(* IEC 61131-3 sources: AXOpen/src/timers/ctrl/test, 4 files *)

(* ---- Abstractions.st ---- *)
USING AxUnit;
USING AXOpen.Timers;
USING AXOpen.Rtc;
USING AXOpen.Logging;
USING AXOpen.Core;
USING AXOpen.Rtc;
USING AXOpen.Rtm;

NAMESPACE AXOpen.Timers_tests

    {S7.extern=ReadWrite}
    CLASS INTERNAL _NULL_LOGGER IMPLEMENTS IAxoLogger
        METHOD PUBLIC Log
            VAR_INPUT
                _message : STRING[80];
                _level : eLogLevel;
                _sender : IAxoObject;
            END_VAR
            ;
        END_METHOD

        METHOD PUBLIC Log
            VAR_INPUT
                _message : STRING[80];
                _level : eLogLevel;
            END_VAR
            ;
        END_METHOD

        METHOD PUBLIC SetMinimumLevel : IAxoLoggerConfig
            VAR_INPUT
                _level : eLogLevel;
            END_VAR
            ;
        END_METHOD
    END_CLASS

    {S7.extern=ReadWrite}
    CLASS INTERNAL AxoRtmMock IMPLEMENTS IAxoRtm
        VAR PRIVATE
            _elapsed : LTIME;
        END_VAR

        METHOD INTERNAL SetElapsed : LDATE_AND_TIME
            VAR_INPUT
                Set :  LTIME;
            END_VAR;
            _elapsed := Set;
        END_METHOD

        METHOD PUBLIC Elapsed : LTIME
            Elapsed := _elapsed;
        END_METHOD
    END_CLASS

    {S7.extern=ReadWrite}
    CLASS INTERNAL TestContext IMPLEMENTS IAxoContext
        VAR PROTECTED
            _openCounter : ULINT;
            _closeCounter : ULINT;
            _identityCounter : ULINT;
            _rtc :  IAxoRtc;
            _rtm :  IAxoRtm;
         END_VAR
        METHOD PUBLIC Open : ULINT
            _openCounter := _openCounter + ULINT#1;
        END_METHOD

        METHOD PUBLIC Close : ULINT
            _closeCounter := _closeCounter + ULINT#1;
        END_METHOD

        METHOD PUBLIC OpenCycleCount : ULINT
            OpenCycleCount := _openCounter;
        END_METHOD

        METHOD PUBLIC ClosedCycleCount : ULINT
            ClosedCycleCount := _closeCounter;
        END_METHOD

        METHOD PUBLIC CreateIdentity : ULINT
            _identityCounter := _identityCounter + ULINT#1;
            CreateIdentity := _identityCounter;
        END_METHOD

        METHOD PUBLIC GetRtc : IAxoRtc ;
            GetRtc := _rtc;
        END_METHOD

        METHOD PUBLIC InjectRtc
             VAR_INPUT Rtc : IAxoRtc;
            END_VAR ;

            _rtc := Rtc;
        END_METHOD

        VAR PRIVATE
            NULL_LOGGER : _NULL_LOGGER;
        END_VAR
        METHOD PUBLIC GetLogger : AXOpen.Logging.IAxoLogger GetLogger := NULL_LOGGER; END_METHOD
        METHOD PUBLIC InjectLogger VAR_INPUT _logger : AXOpen.Logging.IAxoLogger; END_VAR ; END_METHOD

        METHOD PUBLIC GetRtm : IAxoRtm GetRtm := _rtm; END_METHOD
        METHOD PUBLIC InjectRtm VAR_INPUT inRtm : IAxoRtm; END_VAR _rtm := inRtm; END_METHOD
    END_CLASS
END_NAMESPACE

(* ---- OffDelayTests.st ---- *)
USING AxUnit;
USING AXOpen.Timers;
USING AXOpen.Rtc;
USING AXOpen.Logging;
USING AXOpen.Core;
USING AXOpen.Rtc;

NAMESPACE AXOpen.Timers_tests

    {TestFixture}
    {S7.extern=ReadWrite}
    CLASS AxoOffDelayTimersTests
        VAR PROTECTED
            _context : TestContext;
            _inspectedBool : BOOL;
            _rtcMock :  AxoRtmMock;
            _signal : BOOL;
            _testTimerOnDelay: AXOpen.Timers.OnDelayTimer;
            _testTimerOffDelay: AXOpen.Timers.OffDelayTimer;
            _testTimeDelay: LTIME := LTIME#5s;
        END_VAR

        METHOD PRIVATE Initialize
            _context.InjectRtm(_rtcMock);
        END_METHOD

        VAR
            _contextBlank : TestContext;
            _testTimerOnDelayBlank: AXOpen.Timers.OnDelayTimer;
            _testTimerOffDelayBlank: AXOpen.Timers.OffDelayTimer;
        END_VAR

        {TestSetup}
        METHOD PUBLIC TestSetup
        // Will be called before MyTest_A AND before Test_B are executed
            _context := _contextBlank;
            _testTimerOnDelay := _testTimerOnDelayBlank;
            _testTimerOffDelay := _testTimerOffDelayBlank;
        END_METHOD

        {TestTearDown}
        METHOD PUBLIC TestTearDown
        // Will be called after MyTest_A AND before Test_B where executed
            ;
        END_METHOD

        {FixtureSetup}
        METHOD PUBLIC FixtureSetup
        // Will be called once before the Tests are executed
            ;
        END_METHOD

        {FixtureTearDown}
        METHOD PUBLIC FixtureTearDown
        // Will be called after the Tests where executed
            ;
        END_METHOD

        {Test}
        METHOD PUBLIC Timer_offDelay_class_output_test
            THIS.Initialize();

            _context.Open();

            //_rtcMock.SetElapsed(LT#1980-01-23-13:14:33.123456);
            _rtcMock.SetElapsed(LT#0S);
            _signal := TRUE;
            _testTimerOffDelay.OffDelay(_context, _signal, _testTimeDelay);
            Assert.Equal(TRUE, _testTimerOffDelay.output);

            //move 6 seconds in future, timer stil don't count, true is output
            //_rtcMock.SetNowUTC(LDT#1980-01-23-13:14:39.123456);
            _rtcMock.SetElapsed(LT#6S);
            _testTimerOffDelay.OffDelay(_context, _signal, _testTimeDelay);
            Assert.Equal(TRUE, _testTimerOffDelay.output);

            //here, timer starts count
            //_rtcMock.SetNowUTC(LDT#1980-01-23-13:14:41.123456);
            _rtcMock.SetElapsed(LT#9S);
            _signal := FALSE;
            _testTimerOffDelay.OffDelay(_context, _signal, _testTimeDelay);
            Assert.Equal(TRUE, _testTimerOffDelay.output);

            //here, timer should hit delay and turn off signal
            //_rtcMock.SetNowUTC(LDT#1980-01-23-13:14:46.123456);
            _rtcMock.SetElapsed(LT#14S);
            _testTimerOffDelay.OffDelay(_context, _signal, _testTimeDelay);
            Assert.Equal(FALSE, _testTimerOffDelay.output);

            _context.Close();
        END_METHOD

        {Test}
        METHOD PUBLIC Timer_offDelay_overall_test
            THIS.Initialize();

            _context.Open();

            //all turn off, previous signal was false, input is false, output should be false
            //_rtcMock.SetNowUTC(LDT#1980-01-23-13:14:30.0);
            _rtcMock.SetElapsed(LT#10S);
            _signal := FALSE;
            _testTimerOffDelay.OffDelay(_context, _signal, _testTimeDelay);
            Assert.Equal(FALSE, _testTimerOffDelay.output);

            //after 1 second, turn on signal, output should be on
            //_rtcMock.SetNowUTC(LDT#1980-01-23-13:14:31.0);
            _rtcMock.SetElapsed(LT#11S);
            _signal := TRUE;
            _testTimerOffDelay.OffDelay(_context, _signal, _testTimeDelay);
            Assert.Equal(TRUE, _testTimerOffDelay.output);

            //after 2 second, turn off signal, FALLING EDGE detected, output should be on, timer should start counting
            //_rtcMock.SetNowUTC(LDT#1980-01-23-13:14:32.0);
            _rtcMock.SetElapsed(LT#12S);
            _signal := FALSE;
            _testTimerOffDelay.OffDelay(_context, _signal, _testTimeDelay);
            Assert.Equal(TRUE, _testTimerOffDelay.output);

            //after 7 second, timer count passed delay, output should be false
            //_rtcMock.SetNowUTC(LDT#1980-01-23-13:14:35.0);
            _rtcMock.SetElapsed(LT#15S);
            _testTimerOffDelay.OffDelay(_context, _signal, _testTimeDelay);
            Assert.Equal(FALSE, _testTimerOffDelay.output);

            //after 10 second, rising edge was detected, timer is reseted and output should be true
            //_rtcMock.SetNowUTC(LDT#1980-01-23-13:14:40.0);
            _rtcMock.SetElapsed(LT#20S);
            _signal := TRUE;
            _testTimerOffDelay.OffDelay(_context, _signal, _testTimeDelay);
            Assert.Equal(TRUE, _testTimerOffDelay.output);

            //after 11 second, falling edge was detected, timer should start count again
            //_rtcMock.SetNowUTC(LDT#1980-01-23-13:14:41.0);
            _rtcMock.SetElapsed(LT#21S);
            _signal := FALSE;
           _testTimerOffDelay.OffDelay(_context, _signal, _testTimeDelay);
            Assert.Equal(TRUE, _testTimerOffDelay.output);

            //after 13 second, rising edge was detected, timer is reseted, output is still true
            //_rtcMock.SetNowUTC(LDT#1980-01-23-13:14:43.0);
            _rtcMock.SetElapsed(LT#23S);
            _signal := TRUE;
            _testTimerOffDelay.OffDelay(_context, _signal, _testTimeDelay);
            Assert.Equal(TRUE, _testTimerOffDelay.output);

            _context.Close();
        END_METHOD

        {Test}
        METHOD PUBLIC Timer_offDelay_method_output_test
            VAR_TEMP
                _methodOutput: BOOL;
            END_VAR
            THIS.Initialize();

            _context.Open();

            //_rtcMock.SetNowUTC(LDT#1980-01-23-13:14:33.123456);
            _rtcMock.SetElapsed(LT#33S);
            _signal := TRUE;
            _methodOutput := _testTimerOffDelay.OffDelay(_context, _signal, _testTimeDelay);
            Assert.Equal(TRUE, _methodOutput);

            //move 6 seconds in future, timer stil don't count, true is output
            //_rtcMock.SetNowUTC(LDT#1980-01-23-13:14:39.123456);
            _rtcMock.SetElapsed(LT#39S);
            _methodOutput := _testTimerOffDelay.OffDelay(_context, _signal, _testTimeDelay);
            Assert.Equal(TRUE, _methodOutput);

            //here, timer starts count
            //_rtcMock.SetNowUTC(LDT#1980-01-23-13:14:41.123456);
            _rtcMock.SetElapsed(LT#41S);
            _signal := FALSE;
            _methodOutput := _testTimerOffDelay.OffDelay(_context, _signal, _testTimeDelay);
            Assert.Equal(TRUE, _methodOutput);

            //here, timer should hit delay and turn off signal
            //_rtcMock.SetNowUTC(LDT#1980-01-23-13:14:46.123456);
            _rtcMock.SetElapsed(LT#46S);
            _methodOutput := _testTimerOffDelay.OffDelay(_context, _signal, _testTimeDelay);
            Assert.Equal(FALSE, _methodOutput);

            _context.Close();
        END_METHOD

        {Test}
        METHOD PUBLIC Timer_offDelay_delay_is_not_reached_output_is_true
            VAR_TEMP
                _methodOutput: BOOL;
            END_VAR
            THIS.Initialize();

            _context.Open();

            //_rtcMock.SetNowUTC(LDT#1980-01-23-13:14:33.123456);
            _rtcMock.SetElapsed(LT#33S);
            _signal := TRUE;
            _methodOutput := _testTimerOffDelay.OffDelay(_context, _signal, _testTimeDelay);
            Assert.Equal(TRUE, _methodOutput);

            //move 3 seconds in future
            //_rtcMock.SetNowUTC(LDT#1980-01-23-13:14:36.123456);
            _rtcMock.SetElapsed(LT#36S);
            _methodOutput := _testTimerOffDelay.OffDelay(_context, _signal, _testTimeDelay);
            Assert.Equal(TRUE, _methodOutput);

            _context.Close();
        END_METHOD

        {Test}
        METHOD PUBLIC Timer_offDelay_zero_delay
            VAR_TEMP
                _resultET : BOOL;
            END_VAR
            THIS.Initialize();

            //arange
            _context.Open();
            _testTimeDelay := LT#0s;
            //_rtcMock.SetNowUTC(LDT#1980-01-23-13:14:33.123456);
            _rtcMock.SetElapsed(LT#33S);
            _signal := TRUE;

            //act/assert
            _testTimerOffDelay.OffDelay(_context, _signal, _testTimeDelay);
            Assert.Equal(TRUE, _testTimerOffDelay.output);

            _context.Close();
        END_METHOD

        {Test}
        METHOD PUBLIC Timer_offDelay_evertyhing_off
            VAR_TEMP
                _resultET : BOOL;
            END_VAR
            THIS.Initialize();

            //arange
            _context.Open();

            //_rtcMock.SetNowUTC(LDT#1980-01-23-13:14:33.123456);
            _rtcMock.SetElapsed(LT#33S);
            _signal := FALSE;

            //act/assert
            _testTimerOffDelay.OffDelay(_context, _signal, _testTimeDelay);
            Assert.Equal(FALSE, _testTimerOffDelay.output);

            _context.Close();
        END_METHOD

       END_CLASS
END_NAMESPACE

(* ---- OnDelayTests.st ---- *)
USING AxUnit;
USING AXOpen.Timers;
USING AXOpen.Rtc;
USING AXOpen.Logging;
USING AXOpen.Core;
USING AXOpen.Rtc;

NAMESPACE AXOpen.Timers_tests

    {TestFixture}
    {S7.extern=ReadWrite}
    CLASS AxoOnDelayTimersTests
        VAR PROTECTED
            _context : TestContext;
            _inspectedBool : BOOL;
            _rtcMock :  AxoRtcMock;
            _signal : BOOL;
            _testTimerOnDelay: AXOpen.Timers.OnDelayTimer;
            _testTimeDelay: LTIME := LTIME#5s;
        END_VAR

        METHOD PRIVATE Initialize
            _context.InjectRtc(_rtcMock);
        END_METHOD

        VAR
            _contextBlank : TestContext;
            _testTimerOnDelayBlank: AXOpen.Timers.OnDelayTimer;
            _testTimerOffDelayBlank: AXOpen.Timers.OffDelayTimer;
        END_VAR

        {TestSetup}
        METHOD PUBLIC TestSetup
        // Will be called before MyTest_A AND before Test_B are executed
            _context := _contextBlank;
            _testTimerOnDelay := _testTimerOnDelayBlank;
        END_METHOD

        {TestTearDown}
        METHOD PUBLIC TestTearDown
        // Will be called after MyTest_A AND before Test_B where executed
            ;
        END_METHOD

        {FixtureSetup}
        METHOD PUBLIC FixtureSetup
        // Will be called once before the Tests are executed
            ;
        END_METHOD

        {FixtureTearDown}
        METHOD PUBLIC FixtureTearDown
        // Will be called after the Tests where executed
            ;
        END_METHOD

        {Test}
        METHOD PUBLIC Timer_onDelay_overall_test
            THIS.Initialize();

            _context.Open();

            //all turn off, previous signal was false, input is false, output should be false
            _rtcMock.SetNowUTC(LDT#1980-01-23-13:14:30.0);
            _signal := FALSE;
            _testTimerOnDelay.OnDelay(_context, _signal, _testTimeDelay);
            Assert.Equal(FALSE, _testTimeronDelay.output);

            //after 1 second, turn on signal, RISING EDGE detected, counter should start counting, output is still false
            _rtcMock.SetNowUTC(LDT#1980-01-23-13:14:31.0);
            _signal := TRUE;
            _testTimerOnDelay.OnDelay(_context, _signal, _testTimeDelay);
            Assert.Equal(FALSE, _testTimerOnDelay.output);

            //after 6 second, time delay is counted, output should be on
            _rtcMock.SetNowUTC(LDT#1980-01-23-13:14:36.0);
            _testTimerOnDelay.OnDelay(_context, _signal, _testTimeDelay);
            Assert.Equal(TRUE, _testTimerOnDelay.output);

            //after 7 second, nothing changed, output should be on
            _rtcMock.SetNowUTC(LDT#1980-01-23-13:14:37.0);
            _testTimerOnDelay.OnDelay(_context, _signal, _testTimeDelay);
            Assert.Equal(TRUE, _testTimerOnDelay.output);

            //after 8 second, FALLING edge was detected, timer is reseted and output is FALSE
            _rtcMock.SetNowUTC(LDT#1980-01-23-13:14:38.0);
            _signal := FALSE;
            _testTimerOnDelay.OnDelay(_context, _signal, _testTimeDelay);
            Assert.Equal(FALSE, _testTimerOnDelay.output);

            //after 9 second, nothing changed, output is still off
            _rtcMock.SetNowUTC(LDT#1980-01-23-13:14:39.0);
            _testTimerOnDelay.OnDelay(_context, _signal, _testTimeDelay);
            Assert.Equal(FALSE, _testTimerOnDelay.output);

            //after 10 second, rising edge was detected, timer started count again, output is still FALSE
            _rtcMock.SetNowUTC(LDT#1980-01-23-13:14:40.0);
            _signal := TRUE;
            _testTimerOnDelay.OnDelay(_context, _signal, _testTimeDelay);
            Assert.Equal(FALSE, _testTimerOnDelay.output);

            //after 13 second, falling edge was detected, timer was reseted, output is still FALSE
            _rtcMock.SetNowUTC(LDT#1980-01-23-13:14:43.0);
            _signal := FALSE;
            _testTimerOnDelay.OnDelay(_context, _signal, _testTimeDelay);
            Assert.Equal(FALSE, _testTimerOnDelay.output);

            _context.Close();
        END_METHOD

        {Test}
        METHOD PUBLIC Timer_onDelay_class_output_test
            THIS.Initialize();

            //arrange
            _context.Open();
            _rtcMock.SetNowUTC(LDT#1980-01-23-13:14:33.123456);
            _signal := TRUE;

            //act/assert
            _testTimerOnDelay.OnDelay(_context, _signal, _testTimeDelay);
            Assert.Equal(FALSE, _testTimerOnDelay.output);

            //move 6 seconds in future
            _rtcMock.SetNowUTC(LDT#1980-01-23-13:14:39.123456);
            _testTimerOnDelay.OnDelay(_context, _signal, _testTimeDelay);
            Assert.Equal(TRUE, _testTimerOnDelay.output);

            //move 8 seconds in future
            //setting input signal false
            _rtcMock.SetNowUTC(LDT#1980-01-23-13:14:41.123456);
            _signal := FALSE;
            _testTimerOnDelay.OnDelay(_context, _signal, _testTimeDelay);
            Assert.Equal(FALSE, _testTimerOnDelay.output);

            _context.Close();
        END_METHOD

        {Test}
        METHOD PUBLIC Timer_onDelay_method_output_test

            VAR_TEMP
                _methodOutput : BOOL;
            END_VAR
            THIS.Initialize();

            //arange
            _context.Open();
            _rtcMock.SetNowUTC(LDT#1980-01-23-13:14:33.123456);
            _signal := TRUE;

            //act/assert
            _methodOutput := _testTimerOnDelay.OnDelay(_context, _signal, _testTimeDelay);
            Assert.Equal(FALSE, _methodOutput);

            //move 6 seconds in future
            _rtcMock.SetNowUTC(LDT#1980-01-23-13:14:39.123456);
            _methodOutput := _testTimerOnDelay.OnDelay(_context, _signal, _testTimeDelay);
            Assert.Equal(TRUE, _methodOutput);

            //move 8 seconds in future
            //setting input signal false
            _rtcMock.SetNowUTC(LDT#1980-01-23-13:14:41.123456);
            _signal := FALSE;
            _methodOutput := _testTimerOnDelay.OnDelay(_context, _signal, _testTimeDelay);
            Assert.Equal(FALSE, _methodOutput);

            _context.Close();
        END_METHOD

        {Test}
        METHOD PUBLIC Timer_onDelay_delay_is_not_reached_test
            THIS.Initialize();

            //arrange
            _context.Open();
            _rtcMock.SetNowUTC(LDT#1980-01-23-13:14:33.123456);
            _signal := TRUE;

            //act/assert
            _testTimerOnDelay.OnDelay(_context, _signal, _testTimeDelay);
            Assert.Equal(FALSE, _testTimerOnDelay.output);

            //move 2 seconds in future
            _rtcMock.SetNowUTC(LDT#1980-01-23-13:14:35.123456);
            _testTimerOnDelay.OnDelay(_context, _signal, _testTimeDelay);
            Assert.Equal(FALSE, _testTimerOnDelay.output);

            _context.Close();
        END_METHOD

        {Test}
        METHOD PUBLIC Timer_onDelay_class_output_setting_input_signal_false
            THIS.Initialize();

            //arrange
            _context.Open();

            _rtcMock.SetNowUTC(LDT#1980-01-23-13:14:33.123456);
            _signal := TRUE;

            //act/assert
            _testTimerOnDelay.OnDelay(_context, _signal, _testTimeDelay);
            Assert.Equal(FALSE, _testTimerOnDelay.output);

            //move 8 seconds in future
            //setting input signal false
            _rtcMock.SetNowUTC(LDT#1980-01-23-13:14:41.123456);
            _signal := FALSE;
            _testTimerOnDelay.OnDelay(_context, _signal, _testTimeDelay);
            Assert.Equal(FALSE, _testTimerOnDelay.output);

            _context.Close();
        END_METHOD

        {Test}
        METHOD PUBLIC Timer_onDelay_elapsed_time_not_empty
            VAR_TEMP
                _resultET : BOOL;
            END_VAR
            THIS.Initialize();
            //arrange
            _context.Open();
            _rtcMock.SetNowUTC(LDT#1980-01-23-13:14:33.123456);
            _signal := TRUE;

            //act/assert
            _testTimerOnDelay.OnDelay(_context, _signal, _testTimeDelay);
            Assert.Equal(FALSE, _testTimerOnDelay.output);

            //move 7 seconds in future
            _rtcMock.SetNowUTC(LDT#1980-01-23-13:14:40.123456);
            _testTimerOnDelay.OnDelay(_context, _signal, _testTimeDelay);
            _resultET := ((LTIME#7s) = _testTimerOnDelay.elapsedTime);
            Assert.Equal(TRUE, _testTimerOnDelay.output);
            Assert.Equal(TRUE, _resultET);

            _context.Close();
        END_METHOD

        {Test}
        METHOD PUBLIC Timer_onDelay_zero_delay
            VAR_TEMP
                _resultET : BOOL;
            END_VAR
            THIS.Initialize();

            //arange
            _context.Open();
            _testTimeDelay := LT#0s;
            _rtcMock.SetNowUTC(LDT#1980-01-23-13:14:33.123456);
            _signal := TRUE;

            //act/assert
            _testTimerOnDelay.OnDelay(_context, _signal, _testTimeDelay);
            Assert.Equal(TRUE, _testTimerOnDelay.output);

            _context.Close();
        END_METHOD

       END_CLASS
END_NAMESPACE

(* ---- PulseTests.st ---- *)
USING AxUnit;
USING AXOpen.Timers;
USING AXOpen.Rtc;
USING AXOpen.Logging;
USING AXOpen.Core;
USING AXOpen.Rtc;

NAMESPACE AXOpen.Timers_tests

    {TestFixture}
    {S7.extern=ReadWrite}
    CLASS AxoPulseTimersTests
        VAR PROTECTED
            _context : TestContext;
            _inspectedBool : BOOL;
            _rtmMock :  AxoRtmMock;
            _signal : BOOL;
            _testTimerPulse: AXOpen.Timers.PulseTimer;
            _pulseLength: LTIME := LTIME#5s;
        END_VAR

        METHOD PRIVATE Initialize
            _context.InjectRtm(_rtmMock);
        END_METHOD

        {Test}
        METHOD PUBLIC Timer_Pulse_overall_test
            THIS.Initialize();

            _context.Open();

            //all turn off, previous signal was false, input is false, output should be false
            //_rtmMock.SetNowUTC(LDT#1980-01-23-13:14:30.0);
            _rtmMock.SetElapsed(LT#30S);
            _signal := FALSE;
            _testTimerPulse.Pulse(_context, _signal, _pulseLength);
            Assert.Equal(FALSE, _testTimerPulse.output);

            //after 1 second, turn on signal, RISING EDGE detected, counter should start counting, output is still false
            //_rtmMock.SetNowUTC(LDT#1980-01-23-13:14:31.0);
            _rtmMock.SetElapsed(LT#31S);
            _signal := TRUE;
            _testTimerPulse.Pulse(_context, _signal, _pulseLength);
            Assert.Equal(TRUE, _testTimerPulse.output);

            //after 2 second, counting continues, output is still true
            //_rtmMock.SetNowUTC(LDT#1980-01-23-13:14:32.0);
            _rtmMock.SetElapsed(LT#32S);
            _testTimerPulse.Pulse(_context, _signal, _pulseLength);
            Assert.Equal(TRUE, _testTimerPulse.output);

            //after 6 second, pulse length is counted, output will turn off
            //_rtmMock.SetNowUTC(LDT#1980-01-23-13:14:36.0);
            _rtmMock.SetElapsed(LT#36S);
            _testTimerPulse.Pulse(_context, _signal, _pulseLength);
            Assert.Equal(FALSE, _testTimerPulse.output);

            //after 7 second, nothing changed, output should be off
            //_rtmMock.SetNowUTC(LDT#1980-01-23-13:14:37.0);
            _rtmMock.SetElapsed(LT#37S);
            _testTimerPulse.Pulse(_context, _signal, _pulseLength);
            Assert.Equal(FALSE, _testTimerPulse.output);

            //after 8 second, FALLING edge was detected, and timer is counted, therefore is reseted, output is false
            //_rtmMock.SetNowUTC(LDT#1980-01-23-13:14:38.0);
            _rtmMock.SetElapsed(LT#38S);
            _signal := FALSE;
            _testTimerPulse.Pulse(_context, _signal, _pulseLength);
            Assert.Equal(FALSE, _testTimerPulse.output);

            // //after 9 second, nothing changed, output is still off
            // _rtcMock.SetNowUTC(LDT#1980-01-23-13:14:39.0);
            // _testTimerOnDelay.OnDelay(_context, _signal, _testTimeDelay);
            // Assert.Equal(FALSE, _testTimerOnDelay.output);

            // //after 10 second, rising edge was detected, timer started count again, output is still FALSE
            // _rtcMock.SetNowUTC(LDT#1980-01-23-13:14:40.0);
            // _signal := TRUE;
            // _testTimerOnDelay.OnDelay(_context, _signal, _testTimeDelay);
            // Assert.Equal(FALSE, _testTimerOnDelay.output);

            // //after 13 second, falling edge was detected, timer was reseted, output is still FALSE
            // _rtcMock.SetNowUTC(LDT#1980-01-23-13:14:43.0);
            // _signal := FALSE;
            // _testTimerOnDelay.OnDelay(_context, _signal, _testTimeDelay);
            // Assert.Equal(FALSE, _testTimerOnDelay.output);

            _context.Close();
        END_METHOD

       END_CLASS
END_NAMESPACE
